PROGRAM MAIN
VAR
	//bemeneti valtozok
		//fulke ajto jelado
	i_bFulkeNYILT : BOOL;
	i_bFulkeZART : BOOL;
	
		//szintjelzok
	i_bSzintjelzo : ARRAY[0..10] OF BOOL;
	 
		//hivo gombok fel
	i_bHivogombFEL : ARRAY[0..9] OF  BOOL;
		
		//hivo gombok le
	i_bHivogombLE : ARRAY[1..10] OF BOOL;
	
		//fulke gombok (ahova menni akarsz)
	i_bFulkegomb : ARRAY[0..10] OF BOOL; 
	
	//kimeneti valtozok
		//motorok
	q_bFulkeFEL : BOOL;
	q_bFulkeLE : BOOL;
	q_bFulkeNYIT : BOOL;
	q_bFulkeZAR : BOOL;

		//hivo lampak fel
	q_bHivolampaFEL : ARRAY[0..9] OF BOOL;
	
		//hivo lampak le
	q_bHivolampaLE : ARRAY[1..10] OF BOOL; 
	
		//fulkegomb lampak
	q_bFulkegomblampa : ARRAY[0..10] OF BOOL;
	
	//seged valtozok
	nCelEmelet : INT;
	nJelenlegiEmelet : INT;
	
	//timerek
	Ajtomozgas : TON;
END_VAR

//cel emelet regisztralasa
IF i_bHivogombFEL[0] OR i_bFulkegomb[0] THEN
	nCelEmelet := 0;
END_IF

IF i_bHivogombFEL[1] OR i_bHivogombLE[1] OR i_bFulkegomb[1] THEN
	nCelEmelet := 1;
END_IF

IF i_bHivogombFEL[2] OR i_bHivogombLE[2] OR i_bFulkegomb[2] THEN
	nCelEmelet := 2;
END_IF

IF i_bHivogombFEL[3] OR i_bHivogombLE[3] OR i_bFulkegomb[3] THEN
	nCelEmelet := 3;
END_IF

IF i_bHivogombFEL[4] OR i_bHivogombLE[4] OR i_bFulkegomb[4] THEN
	nCelEmelet := 4;
END_IF

IF i_bHivogombFEL[5] OR i_bHivogombLE[5] OR i_bFulkegomb[5] THEN
	nCelEmelet := 5;
END_IF

IF i_bHivogombFEL[6] OR i_bHivogombLE[6] OR i_bFulkegomb[6] THEN
	nCelEmelet := 6;
END_IF

IF i_bHivogombFEL[7] OR i_bHivogombLE[7] OR i_bFulkegomb[7] THEN
	nCelEmelet := 7;
END_IF

IF i_bHivogombFEL[8] OR i_bHivogombLE[8] OR i_bFulkegomb[8] THEN
	nCelEmelet := 8;
END_IF

IF i_bHivogombFEL[9] OR i_bHivogombLE[9] OR i_bFulkegomb[9] THEN
	nCelEmelet := 9;
END_IF

IF i_bHivogombLE[10] OR i_bFulkegomb[10] THEN
	nCelEmelet := 10;
END_IF

//fulke megerkezes eszlelese
IF nCelemelet = 0 AND i_bSzintjelzo[0] THEN
	nJelenlegiEmelet := nCelEmelet;
END_IF

IF nCelemelet = 1 AND i_bSzintjelzo[1] THEN
	nJelenlegiEmelet := nCelEmelet;
END_IF

IF nCelemelet = 2 AND i_bSzintjelzo[2] THEN
	nJelenlegiEmelet := nCelEmelet;
END_IF

IF nCelemelet = 3 AND i_bSzintjelzo[3] THEN
	nJelenlegiEmelet := nCelEmelet;
END_IF

IF nCelemelet = 4 AND i_bSzintjelzo[4]THEN
	nJelenlegiEmelet := nCelEmelet;
END_IF

IF nCelemelet = 5 AND i_bSzintjelzo[5] THEN
	nJelenlegiEmelet := nCelEmelet;
END_IF

IF nCelemelet = 6 AND i_bSzintjelzo[6] THEN
	nJelenlegiEmelet := nCelEmelet;
END_IF

IF nCelemelet = 7 AND i_bSzintjelzo[7] THEN
	nJelenlegiEmelet := nCelEmelet;
END_IF

IF nCelemelet = 8 AND i_bSzintjelzo[8] THEN
	nJelenlegiEmelet := nCelEmelet;
END_IF

IF nCelemelet = 9 AND i_bSzintjelzo[9] THEN
	nJelenlegiEmelet := nCelEmelet;
END_IF

IF nCelemelet = 10 AND i_bSzintjelzo[10] THEN
	nJelenlegiEmelet := nCelEmelet;
END_IF

//ajto nyitas megadasa
IF (nJelenlegiEmelet = nCelEmelet) AND NOT (q_bFulkeFEL OR q_bFulkeLE) THEN
	q_bFulkeNYIT := TRUE;
	ELSIF q_bFulkeFEL OR q_bFulkeLE THEN
		q_bFulkeNYIT := FALSE;
	ELSE
		q_bFulkeNYIT := FALSE;
END_IF

//ajto zaras megadasa -- talan teljesen kihagyhato es megadhato az ajtonyitas else agaban?
IF (nJelenlegiEmelet <> nCelEmelet) AND NOT (q_bFulkeFEL OR q_bFulkeLE) THEN
	q_bFulkeZAR := TRUE;
	ELSE
		q_bFulkeZAR := FALSE;
END_IF

//gomb megnyomas es lampa felgyulladas osszekotese 
	//hivo gombok fel	
IF i_bHivogombFEL[0] THEN
	q_bHivolampaFEL[0] := TRUE;
	ELSIF nCelEmelet = nJelenlegiEmelet AND NOT i_bFulkeZART THEN
		q_bHivolampaFEL[0] := FALSE;
	ELSE
		q_bHivolampaFEL[0] := FALSE;	
END_IF

IF i_bHivogombFEL[1] THEN
	q_bHivolampaFEL[1] := TRUE;
		ELSIF nCelEmelet = nJelenlegiEmelet AND NOT i_bFulkeZART THEN
		q_bHivolampaFEL[1] := FALSE;
	ELSE
		q_bHivolampaFEL[1] := FALSE;	
END_IF

IF i_bHivogombFEL[2] THEN
	q_bHivolampaFEL[2] := TRUE;
		ELSIF nCelEmelet = nJelenlegiEmelet AND NOT i_bFulkeZART THEN
		q_bHivolampaFEL[2] := FALSE;
	ELSE
		q_bHivolampaFEL[2] := FALSE;	
END_IF

IF i_bHivogombFEL[3] THEN
	q_bHivolampaFEL[3] := TRUE;
		ELSIF nCelEmelet = nJelenlegiEmelet AND NOT i_bFulkeZART THEN
		q_bHivolampaFEL[3] := FALSE;
	ELSE
		q_bHivolampaFEL[3] := FALSE;	
END_IF

IF i_bHivogombFEL[4] THEN
	q_bHivolampaFEL[4] := TRUE;
		ELSIF nCelEmelet = nJelenlegiEmelet AND NOT i_bFulkeZART THEN
		q_bHivolampaFEL[4] := FALSE;
	ELSE
		q_bHivolampaFEL[4] := FALSE;	
END_IF

IF i_bHivogombFEL[5] THEN
	q_bHivolampaFEL[5] := TRUE;
		ELSIF nCelEmelet = nJelenlegiEmelet AND NOT i_bFulkeZART THEN
		q_bHivolampaFEL[5] := FALSE;
	ELSE
		q_bHivolampaFEL[5] := FALSE;	
END_IF

IF i_bHivogombFEL[6] THEN
	q_bHivolampaFEL[6] := TRUE;
		ELSIF nCelEmelet = nJelenlegiEmelet AND NOT i_bFulkeZART THEN
		q_bHivolampaFEL[6] := FALSE;
	ELSE
		q_bHivolampaFEL[6] := FALSE;	
END_IF

IF i_bHivogombFEL[7] THEN
	q_bHivolampaFEL[7] := TRUE;
		ELSIF nCelEmelet = nJelenlegiEmelet AND NOT i_bFulkeZART THEN
		q_bHivolampaFEL[7] := FALSE;
	ELSE
		q_bHivolampaFEL[7] := FALSE;	
END_IF

IF i_bHivogombFEL[8] THEN
	q_bHivolampaFEL[8] := TRUE;
		ELSIF nCelEmelet = nJelenlegiEmelet AND NOT i_bFulkeZART THEN
		q_bHivolampaFEL[8] := FALSE;
	ELSE
		q_bHivolampaFEL[8] := FALSE;	
END_IF

IF i_bHivogombFEL[9] THEN
	q_bHivolampaFEL[9] := TRUE;
		ELSIF nCelEmelet = nJelenlegiEmelet AND NOT i_bFulkeZART THEN
		q_bHivolampaFEL[8] := FALSE;
	ELSE
		q_bHivolampaFEL[8] := FALSE;	
END_IF

	//hivo gombok le
IF i_bHivogombLE[1] THEN
	q_bHivolampaLE[1] := TRUE;
	ELSIF nCelEmelet = nJelenlegiEmelet AND NOT i_bFulkeZART THEN
		q_bHivolampaLE[1] := FALSE;
	ELSE
		q_bHivolampaLE[1] := FALSE;	
END_IF

IF i_bHivogombLE[2] THEN
	q_bHivolampaLE[2] := TRUE;
	ELSIF nCelEmelet = nJelenlegiEmelet AND NOT i_bFulkeZART THEN
		q_bHivolampaLE[2] := FALSE;
	ELSE
		q_bHivolampaLE[2] := FALSE;	
END_IF

IF i_bHivogombLE[3] THEN
	q_bHivolampaLE[3] := TRUE;
	ELSIF nCelEmelet = nJelenlegiEmelet AND NOT i_bFulkeZART THEN
		q_bHivolampaLE[3] := FALSE;
	ELSE
		q_bHivolampaLE[3] := FALSE;	
END_IF

IF i_bHivogombLE[4] THEN
	q_bHivolampaLE[4] := TRUE;
	ELSIF nCelEmelet = nJelenlegiEmelet AND NOT i_bFulkeZART THEN
		q_bHivolampaLE[4] := FALSE;
	ELSE
		q_bHivolampaLE[4] := FALSE;	
END_IF

IF i_bHivogombLE[5] THEN
	q_bHivolampaLE[5] := TRUE;
	ELSIF nCelEmelet = nJelenlegiEmelet AND NOT i_bFulkeZART THEN
		q_bHivolampaLE[5] := FALSE;
	ELSE
		q_bHivolampaLE[5] := FALSE;	
END_IF

IF i_bHivogombLE[6] THEN
	q_bHivolampaLE[6] := TRUE;
	ELSIF nCelEmelet = nJelenlegiEmelet AND NOT i_bFulkeZART THEN
		q_bHivolampaLE[6] := FALSE;
	ELSE
		q_bHivolampaLE[6] := FALSE;	
END_IF

IF i_bHivogombLE[7] THEN
	q_bHivolampaLE[7] := TRUE;
	ELSIF nCelEmelet = nJelenlegiEmelet AND NOT i_bFulkeZART THEN
		q_bHivolampaLE[7] := FALSE;
	ELSE
		q_bHivolampaLE[7] := FALSE;	
END_IF

IF i_bHivogombLE[8] THEN
	q_bHivolampaLE[8] := TRUE;
	ELSIF nCelEmelet = nJelenlegiEmelet AND NOT i_bFulkeZART THEN
		q_bHivolampaLE[8] := FALSE;
	ELSE
		q_bHivolampaLE[8] := FALSE;	
END_IF

IF i_bHivogombLE[9] THEN
	q_bHivolampaLE[9] := TRUE;
	ELSIF nCelEmelet = nJelenlegiEmelet AND NOT i_bFulkeZART THEN
		q_bHivolampaLE[9] := FALSE;
	ELSE
		q_bHivolampaLE[9] := FALSE;	
END_IF

IF i_bHivogombLE[10] THEN
	q_bHivolampaLE[10] := TRUE;
	ELSIF nCelEmelet = nJelenlegiEmelet AND NOT i_bFulkeZART THEN
		q_bHivolampaLE[10] := FALSE;
	ELSE
		q_bHivolampaLE[10] := FALSE;	
END_IF

	//fulkegomb lampak
IF i_bFulkegomb[0] THEN
	q_bFulkegomblampa[0] := TRUE;
	ELSIF nCelEmelet = nJelenlegiEmelet AND NOT i_bFulkeZART THEN
		q_bFulkegomblampa[0] := FALSE;
	ELSE
		q_bFulkegomblampa[0] := FALSE;	
END_IF
	
IF i_bFulkegomb[1] THEN
	q_bFulkegomblampa[1] := TRUE;
	ELSIF nCelEmelet = nJelenlegiEmelet AND NOT i_bFulkeZART THEN
		q_bFulkegomblampa[1] := FALSE;
	ELSE
		q_bFulkegomblampa[1] := FALSE;	
END_IF

IF i_bFulkegomb[2] THEN
	q_bFulkegomblampa[2] := TRUE;
	ELSIF nCelEmelet = nJelenlegiEmelet AND NOT i_bFulkeZART THEN
		q_bFulkegomblampa[2] := FALSE;
	ELSE
		q_bFulkegomblampa[2] := FALSE;	
END_IF

IF i_bFulkegomb[3] THEN
	q_bFulkegomblampa[3] := TRUE;
	ELSIF nCelEmelet = nJelenlegiEmelet AND NOT i_bFulkeZART THEN
		q_bFulkegomblampa[3] := FALSE;
	ELSE
		q_bFulkegomblampa[3] := FALSE;	
END_IF

IF i_bFulkegomb[4] THEN
	q_bFulkegomblampa[4] := TRUE;
	ELSIF nCelEmelet = nJelenlegiEmelet AND NOT i_bFulkeZART THEN
		q_bFulkegomblampa[4] := FALSE;
	ELSE
		q_bFulkegomblampa[4] := FALSE;	
END_IF

IF i_bFulkegomb[5] THEN
	q_bFulkegomblampa[5] := TRUE;
	ELSIF nCelEmelet = nJelenlegiEmelet AND NOT i_bFulkeZART THEN
		q_bFulkegomblampa[5] := FALSE;
	ELSE
		q_bFulkegomblampa[5] := FALSE;	
END_IF

IF i_bFulkegomb[6] THEN
	q_bFulkegomblampa[6] := TRUE;
	ELSIF nCelEmelet = nJelenlegiEmelet AND NOT i_bFulkeZART THEN
		q_bFulkegomblampa[6] := FALSE;
	ELSE
		q_bFulkegomblampa[6] := FALSE;	
END_IF

IF i_bFulkegomb[7] THEN
	q_bFulkegomblampa[7] := TRUE;
	ELSIF nCelEmelet = nJelenlegiEmelet AND NOT i_bFulkeZART THEN
		q_bFulkegomblampa[7] := FALSE;
	ELSE
		q_bFulkegomblampa[7] := FALSE;	
END_IF

IF i_bFulkegomb[8] THEN
	q_bFulkegomblampa[8] := TRUE;
	ELSIF nCelEmelet = nJelenlegiEmelet AND NOT i_bFulkeZART THEN
		q_bFulkegomblampa[8] := FALSE;
	ELSE
		q_bFulkegomblampa[8] := FALSE;	
END_IF

IF i_bFulkegomb[9] THEN
	q_bFulkegomblampa[9] := TRUE;
	ELSIF nCelEmelet = nJelenlegiEmelet AND NOT i_bFulkeZART THEN
		q_bFulkegomblampa[9] := FALSE;
	ELSE
		q_bFulkegomblampa[9] := FALSE;	
END_IF

IF i_bFulkegomb[10] THEN
	q_bFulkegomblampa[10] := TRUE;
	ELSIF nCelEmelet = nJelenlegiEmelet AND NOT i_bFulkeZART THEN
		q_bFulkegomblampa[10] := FALSE;
	ELSE
		q_bFulkegomblampa[10] := FALSE;	
END_IF

END_PROGRAM

(* stored: Version 1.1.0.1
   POU MAIN: Id {6ba8dc1c-e289-46b1-bfea-79f9f7b690a7}, SpecialFunc None *)
